PROGRAM MAIN
VAR
	//Variables of type AXIS_REF to your motors.
	//Add more motors if you need to.
	
	motor_x0 : AxisBase;
	motor_y0 : AxisBase;
	motor_z0 : AxisBase;
	motor_a0 : AxisBase;
	motor_b0 : AxisBase;
END_VAR

motor_x0();
motor_y0();
motor_z0();
motor_a0();
motor_b0();


IO();
Recorder();

END_PROGRAM

(* stored: Version 1.1.0.1, ProductVersion 3.1.4024.12
   POU MAIN: Id {34dbeb6e-0188-42c2-aa4f-4993de0a93ee}, SpecialFunc None *)
